{attribute addProperty BoxType "EP6228-3132-0016"}
{attribute addProperty Id "Digital_InputsDigital_Inputs_910A3194324"}
{attribute addProperty CRC "232856839"}
{attribute addProperty SizeInBites "32"}
{attribute addProperty SizeInBytes "4"}
TYPE Module_11_Digital_Inputs_0DE11D07 :
STRUCT
	{attribute addProperty Name "Digital_Inputs"}
	Digital_Inputs  : Digital_Inputs_910A3194;
END_STRUCT
END_TYPE

(* stored: Version 1.2.0.0, ProductVersion 3.1.4024.9
   DUT Module_11_Digital_Inputs_0DE11D07: Id {6650ed03-6a70-4f42-8eb8-aac8b2b2e243} *)
